ABB RobotStudio station: OpenRoboticaISEP2023.rspag

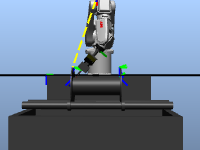
--- station ---
Station station_version_TEst (saved by RobotStudio 7.0.8504.151)
Controller IRB120ob
  mechanical unit ROB_1: IRB120_3_58__01, 6 joints, base frame (0, 0, 0) mm
Layout (positions relative to the parent item):
  - IRB120_3_58__01 [mechanism, from Robots\IRB120_3_58_G_01.rslib] at (0, 0, 0) mm; joint values [0.1437, 0.7309, 0.5088, -1.0759, 0.7904, 1.101] (rad or m)
  - Group_1_5 [graphiccomponentgroup, from Modelos\Garra-OpenRobotica.rslib] at (341.04, 3.87, 172.38) mm, rotated rx -140.81 ry 0 rz 180 deg
    - _SCHUNK-5518814_G10001085_0 [graphiccomponentgroup, from Modelos\Garra-OpenRobotica.rslib] at (0, 0, 60) mm, rotated rx 0 ry 90 rz 0 deg
      - _SCHUNK-5518813_A10001086_0 [graphiccomponentgroup, from Modelos\Garra-OpenRobotica.rslib]
        - _SCHUNK-5518813_F10001087_0 [graphiccomponentgroup, from Modelos\Garra-OpenRobotica.rslib]
          - _SCHUNK-9962715_B10001088_0 [graphiccomponentgroup, from Modelos\Garra-OpenRobotica.rslib]
            - _SCHUNK-9965220-S10001089_0 [part, from Modelos\Garra-OpenRobotica.rslib]
            - _SCHUNK-9962715_B10001088_0 [part, from Modelos\Garra-OpenRobotica.rslib]
          - _SCHUNK-9962715_B10001090_0 [graphiccomponentgroup, from Modelos\Garra-OpenRobotica.rslib]
            - _SCHUNK-9965220-S10001101_0 [part, from Modelos\Garra-OpenRobotica.rslib]
            - _SCHUNK-9962715_B10001090_0 [part, from Modelos\Garra-OpenRobotica.rslib]
          - _SCHUNK-5518813_F10001087_0 [part, from Modelos\Garra-OpenRobotica.rslib]
        - _SCHUNK-5518813_F10001093_0 [graphiccomponentgroup, from Modelos\Garra-OpenRobotica.rslib]
          - _SCHUNK-9962715_B10001094_0 [graphiccomponentgroup, from Modelos\Garra-OpenRobotica.rslib]
            - _SCHUNK-9965220-S10001095_0 [part, from Modelos\Garra-OpenRobotica.rslib]
            - _SCHUNK-9962715_B10001094_0 [part, from Modelos\Garra-OpenRobotica.rslib]
          - _SCHUNK-9962715_B10001096_0 [graphiccomponentgroup, from Modelos\Garra-OpenRobotica.rslib]
            - _SCHUNK-9965220-S10001097_0 [part, from Modelos\Garra-OpenRobotica.rslib]
            - _SCHUNK-9962715_B10001096_0 [part, from Modelos\Garra-OpenRobotica.rslib]
          - _SCHUNK-5518813_F10001093_0 [part, from Modelos\Garra-OpenRobotica.rslib]
        - _SCHUNK-9905502_T10001099_0 [part, from Modelos\Garra-OpenRobotica.rslib]
        - _SCHUNK-5518813_A10001086_0 [part, from Modelos\Garra-OpenRobotica.rslib]
      - _SCHUNK-5518814_G10001085_0 [part, from Modelos\Garra-OpenRobotica.rslib]
    - body [part, from Modelos\Garra-OpenRobotica.rslib] at (0, 0, 238) mm, rotated rx 0 ry 90 rz 0 deg
    - Extensão-Garra [part, from Modelos\Garra-OpenRobotica.rslib] at (0, 0, 0) mm, rotated rx 0 ry 0 rz 90 deg
    - SCHUNK-0340215 ABR-MPG-plus 64_Aluminum [part, from Modelos\Garra-OpenRobotica.rslib] at (0, 0, 178) mm, rotated rx 180 ry 0 rz 90 deg
    - SCHUNK-0340215 ABR-MPG-plus 64_Aluminum_2 [part, from Modelos\Garra-OpenRobotica.rslib] at (0, 0, 178) mm, rotated rx 180 ry 0 rz -90 deg
  - MyNewTool [mechanism, from Tools\tool1.rslib] at (341.04, 3.87, 172.38) mm, rotated rx -140.81 ry 0 rz 180 deg
  - Estrutura [graphiccomponentgroup]
    - Part_15 [part] at (0, 34.25, 13) mm
    - Part_10 [part] at (0, 34.03, 13) mm
    - Part_9 [part] at (0, 32.93, 13) mm
    - Part_8 [part] at (0, 0, 13) mm
    - Part_7 [part] at (0, 0, 13) mm
    - Part_6 [part] at (0, 0, 13) mm
    - Part_3 [part]
Attachment: Group_1_5 is attached to IRB120_3_58__01 / Link6
Attachment: MyNewTool is attached to IRB120_3_58__01 / Link6
Targets, tools, work objects and paths stored in the station and not in the controller backup, written as RAPID:
! task T_ROB1
MODULE Module1
  CONST robtarget target_ref_mesa:=[[132.65,-385.03,4.02],[0,0,1,0],[0,0,0,0],[9E+09,9E+09,9E+09,9E+09,9E+09,9E+09]];
ENDMODULE


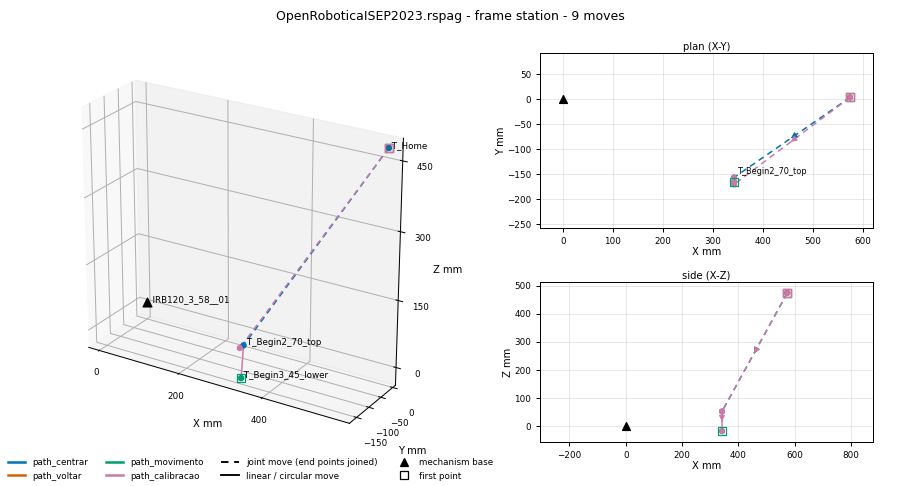
[picture p0: tool path of OpenRoboticaISEP2023.rspag in frame station, 9 of 11 moves have a stored position in this frame; points joined in program order, loops and branches not executed]
--- Backups/IRB120ob/RAPID/TASK1/PROGMOD/CalibData.mod ---
MODULE CalibData
	PERS tooldata tcptool:=[TRUE,[[-1.2328,3.617,241.774],[1,0,0,0]],[1,[0,0,125],[1,0,0,0],0,0,0]];
ENDMODULE

--- Backups/IRB120ob/RAPID/TASK1/PROGMOD/Module1.mod ---
MODULE Module1

    !************************************************!
    !Autores : Fabio Pacheco, Simao Duarte           !
    !                                                !
    !Version: Estado deixado apos o openRobotica2023 !
    !                                                !
    !************************************************!

    !targets-begin
	CONST robtarget T_Home:=[[574.352655047,3.617,474.180636118],[0.5,0,0.866025404,0],[0,-1,0,0],[9E+09,9E+09,9E+09,9E+09,9E+09,9E+09]];

    CONST robtarget T_Begin1_90_top:=[[342.277,-170.47,52.7],[0,0,1,0],[0,0,0,0],[9E+09,9E+09,9E+09,9E+09,9E+09,9E+09]];
	CONST robtarget T_Begin2_70_top:=[[342.277,-156.47,52.7],[0,0,0.984807753,-0.173648178],[0,0,0,0],[9E+09,9E+09,9E+09,9E+09,9E+09,9E+09]];
    CONST robtarget T_Begin3_45_lower:=[[342.277,-165.47,-17.3],[0,0,0.923879533,-0.382683432],[0,0,0,0],[9E+09,9E+09,9E+09,9E+09,9E+09,9E+09]];

    !targets-end-var
    PERS robtarget T_End1_45_lower:=[[342.277,134.53,-17.3],[0,0,0.92388,0.382683],[0,0,0,0],[9E+09,9E+09,9E+09,9E+09,9E+09,9E+09]];
    CONST robtarget T_End2_70_top:=[[342.277,146.6,52.7],[0,0,0.984807753,0.173648177],[0,0,-1,0],[9E+09,9E+09,9E+09,9E+09,9E+09,9E+09]];
    CONST robtarget T_End3_90_top:=[[342.277,149.6,52.7],[0,0,1,0],[0,0,0,0],[9E+09,9E+09,9E+09,9E+09,9E+09,9E+09]];


    !info needed
    !raio do pneu (rp), espessura do cordao (esp), largura do pneu(lp), sobreposiçao (sob)
    !velocidade(v), tempo (rota. completa)->(t), velocidade_x (vx)

        VAR num rp:=-1;
        VAR num esp:=-1;
        VAR num lp:=-1;
        VAR num v:=-1;
        VAR num vx;
        VAR num sob:=-1;

        !opçoes menus
        VAR num menu;
        VAR num menu2;

        CONST num dim_largura_pneu_max := 500;
        CONST num dim_largura_pneu_min := 100;
        CONST num dim_raio_pneu_max := 300;
        CONST num dim_raio_pneu_min := 50;
        CONST num dim_raio_sl_max := 11;
        CONST num dim_raio_sl_min := 1;
        CONST num dim_sob_sl_max := 100;
        CONST num dim_sob_sl_min := 0;
        CONST num v_max := 100;
        CONST num v_min := 0.0353;


    PROC main()

        WHILE menu<>-1 DO !Menu principal

            TPReadFK menu,"Bem-vindo ao menu","START","EDIT-PNEU","EDIT-SILI.","EDIT-VEL.","MAPING";

            IF menu=5 THEN
                !calibration program
                IF rp = -1 OR esp =-1 OR lp = -1 OR v = -1 OR sob = -1 THEN
                    TPWrite "Erro fatal : Necessario corrigir valores.";
                ELSE
                    TPWrite("Teste de calibraçao: (a velocidade do robot sera limitada)");
                    path_calibracao;
                ENDIF
            ELSE
                    IF menu=1 THEN
                        !start program
                        IF rp = -1 OR esp =-1 OR lp = -1 OR v = -1 OR sob = -1 THEN
                            TPWrite "Erro fatal : Necessario corrigir valores.";
                        ELSE
                            !Path_10;
                            path_centrar;
                            path_movimento;
                            path_voltar;
                        ENDIF
                    ELSEIF menu=2 THEN
                        TPReadFK menu2,"Menu para modificar o pneu, escolha.","Raio(mm)","Largura(mm)",stEmpty,stEmpty,"Voltar";

                        !TEST menu2 !menu para especificar os valores de um determinado objeto

                        IF menu2 = 1 THEN
                            !raio
                            TPWrite("Raio do pneu em [50mm - 300mm]");
                            rp:= askVALUE(dim_raio_pneu_min,dim_raio_pneu_max);
                        ElSEIF menu2 = 2 THEN
                            !largura
                            TPWrite("Largura do pneu em [100mm - 500mm]");
                            lp:= askVALUE(dim_largura_pneu_min,dim_largura_pneu_max);
                        ELSEIF menu2 = 5 THEN
                            menu2:=-1;
                        ENDIF


                    ELSEIF menu=3 THEN
                        TPReadFK menu2,"Menu para modificar o silicone, escolha.","Espessura","Sobreposiçao",stEmpty,stEmpty,"Voltar";

                        !TEST menu2 !menu para especificar os valores de um determinado objeto

                        IF menu2 = 1 THEN !espessura
                            !TPWrite "Espessura em ["  + NumToStr(dim_raio_sl_min) + "mm - " + NumToStr(dim_raio_sl_max) + "mm]";
                            TPWrite("Espessura em [1mm - 11mm]");
                            esp:= askVALUE(dim_raio_sl_min,dim_raio_sl_max);
                        ELSEIF menu2 = 2 THEN !sobreposicao
                            TPWrite("Sobreposiçao em [0% - 100%]");
                            sob:= askVALUE(dim_sob_sl_min,dim_sob_sl_max);
                        ELSE
                            menu2:=-1;
                        ENDIF


                    ELSEIF menu=4 THEN
                        !velocidade
                        TPWrite("Velocidade em [1%-100%]");
                        v:= askVALUE(v_min,v_max);
                    ENDIF !main
            ENDIF
        ENDWHILE
    ENDPROC

    FUNC num askVALUE(num min, num max)
        VAR num value:=-1;
        WHILE value < min OR value > max DO
                TPReadNum value, "Qual o valor?";
        ENDWHILE
        RETURN value;
    ENDFUNC

    FUNC num calcVin(num v, num esp, num sob)
        VAR num vx;
        v:=v/100;
        sob:=sob/100;
        vx := ((esp * (1 - sob) * 60 * 0.0125)/(v - 0.0352)); !(m/s)
        RETURN vx;
    ENDFUNC

    PROC path_centrar()
        MoveJ T_Home,v150,z100,tcptool\WObj:=wobj0;
        !MoveJ T_Begin1_90_top,v100,fine,tcptool\WObj:=wobj0;
	    MoveJ T_Begin2_70_top,v100,fine,tcptool\WObj:=wobj0;
    ENDPROC

    PROC path_voltar()
        MoveJ T_Home,v150,z100,tcptool\WObj:=wobj0;
    ENDPROC

    PROC path_movimento()
        VAR speeddata vx := [1,20,500,500];
        vx := [calcVin(v,esp,sob),20,500,500];
        T_End1_45_lower.trans.y:=T_Begin3_45_lower.trans.y+lp;
        MoveL T_Begin3_45_lower,v30,fine,tcptool\WObj:=wobj0;
	    MoveL T_End1_45_lower,vx,fine,tcptool\WObj:=wobj0;
    ENDPROC

    PROC path_calibracao()
        !teste pathing
        VAR speeddata vx := [1,20,500,500];
        vx := [calcVin(v,esp,sob),20,500,500];
        T_End1_45_lower.trans.y:=T_Begin3_45_lower.trans.y+lp;

        MoveJ T_Home,v100,z100,tcptool\WObj:=wobj0;
        MoveJ T_Begin1_90_top,v50,fine,tcptool\WObj:=wobj0;
	    MoveJ T_Begin2_70_top,v30,fine,tcptool\WObj:=wobj0;

        MoveL T_Begin3_45_lower,v10,fine,tcptool\WObj:=wobj0;
	    MoveL T_End1_45_lower,vx,fine,tcptool\WObj:=wobj0;

        MoveJ T_Home,v100,z100,tcptool\WObj:=wobj0;

    ENDPROC
ENDMODULE

--- Backups/IRB120ob/SYSPAR/EIO.cfg ---
EIO:CFG_1.0:5:0::
#
EIO_BUS:

      -Name "Virtual1" -ConnectorID "SIM1"
#
EIO_UNIT_TYPE:

      -Name "Virtual" -VendorName "ABB" -ProductName "Virtual unit"
#
EIO_ACCESS:

      -Name "All" -Rapid  -LocalManual  -LocalAuto  -RemoteManual  -RemoteAuto
